{attribute 'no_explicit_call' := 'do not call this function block directly'} 
FUNCTION_BLOCK ABSTRACT ProgramState EXTENDS ToolkitObject
VAR_OUTPUT
	{attribute 'OPC.UA.DA.Access' := '1'}
	FromTransitions : ARRAY [0..ProgramConstants.MaxTransitionCount - 1] OF STRING;
	{attribute 'OPC.UA.DA.Access' := '1'}
	FromTransitionCount : INT(0..ProgramConstants.MaxTransitionCount - 1);
	{attribute 'OPC.UA.DA.Access' := '1'}
	ToTransitions : ARRAY [0..ProgramConstants.MaxTransitionCount - 1] OF STRING;
	{attribute 'OPC.UA.DA.Access' := '1'}
	ToTransitionCount : INT(0..ProgramConstants.MaxTransitionCount - 1);
END_VAR
VAR
	{attribute 'OPC.UA.DA' := '0'}
	_Busy : BOOL;
	{attribute 'OPC.UA.DA' := '0'}
	_Error : BOOL;

	{attribute 'OPC.UA.DA' := '0'}
	_StateMachine : REFERENCE TO FiniteStateMachine;
END_VAR

{attribute 'monitoring' := 'call'}
{attribute 'OPC.UA.DA.Property' := '1'}
{attribute 'OPC.UA.DA.Access' := '1'}
PROPERTY Busy : BOOL
GET
Busy := _Busy;
END_GET
END_PROPERTY

METHOD Disable
IF _Busy THEN
	_Busy := FALSE;
END_IF
END_METHOD

METHOD Enable
_Busy := TRUE;
_Error := FALSE;
END_METHOD

{attribute 'monitoring' := 'call'}
{attribute 'OPC.UA.DA.Property' := '1'}
{attribute 'OPC.UA.DA.Access' := '1'}
PROPERTY Error : BOOL
GET
Error := _Error;
END_GET
END_PROPERTY

METHOD Execute
END_METHOD

METHOD Initialize 
VAR_INPUT
	stateMachine : REFERENCE TO FiniteStateMachine;
END_VAR
IF NOT __ISVALIDREF(_StateMachine) THEN
	//exceptionFactory.ThrowException(__POSITION(), "programStateMachine is NULL");
END_IF

_StateMachine REF= stateMachine;
END_METHOD

{attribute 'monitoring' := 'call'}
{attribute 'OPC.UA.DA.Property' := '1'}
{attribute 'OPC.UA.DA.Access' := '1'}
PROPERTY Initialized : BOOL
GET
Initialized := __ISVALIDREF(_StateMachine);
END_GET
END_PROPERTY

{attribute 'monitoring' := 'call'}
PROPERTY LastException : REFERENCE TO Exception
GET
LastException REF= _LastException;
END_GET
END_PROPERTY

{attribute 'monitoring' := 'call'}
{attribute 'OPC.UA.DA.Property' := '1'}
{attribute 'OPC.UA.DA.Access' := '1'}
PROPERTY ABSTRACT Name : STRING
GET
END_GET
END_PROPERTY

METHOD INTERNAL FINAL RegisterTransition
VAR_INPUT
	transition : REFERENCE TO ProgramTransition;
END_VAR
IF transition.FromState = Name THEN
	ToTransitions[ToTransitionCount] := transition.Name;
	ToTransitionCount := ToTransitionCount + 1;
ELSIF transition.ToState = Name THEN
	FromTransitions[FromTransitionCount] := transition.Name;
	FromTransitionCount := FromTransitionCount + 1;
END_IF
END_METHOD

END_FUNCTION_BLOCK

(* stored: Version 1.1.0.1
   POU ProgramState: Id {c31cfc44-ae43-4468-b5cf-1bc32fd490b1}, SpecialFunc None
   Property Busy: Id {9a0eb3d2-0b01-4f39-93a4-f08c1588ba3d}
   Get Get: Id {d9c4b9d4-7603-49ff-8edb-0ecfd981ae49}
   Method Disable: Id {7d85a8d6-8ab4-4e70-87c0-c45f5a00e8d1}
   Method Enable: Id {1245c2db-628d-4e38-b794-4908c55fcf8b}
   Property Error: Id {20d253f1-bf46-4081-b875-ca324598e944}
   Get Get: Id {0757b6f6-21a2-4441-ad86-63a98924171c}
   Method Execute: Id {45725f05-e410-43ff-ab0c-e99117c43a9a}
   Method Initialize: Id {c288b58b-ee60-4513-924e-b42e94c3adb4}
   Property Initialized: Id {850bf25a-2c15-4908-9e8c-b1bb1d129764}
   Get Get: Id {610e4bac-7767-4349-9689-40b779b58cd2}
   Property LastException: Id {fd638560-9710-41cd-90ef-077713fec448}
   Get Get: Id {369908df-91c8-4d1f-a005-1f8a4493cb81}
   Property Name: Id {41fdd47d-a30d-4367-b646-356c5a46d9b7}
   Get Get: Id {eced237f-20a3-4c55-afdb-2ca7266e825c}
   Method RegisterTransition: Id {b0f513a5-20d8-444f-95da-0e3e732b074d} *)
